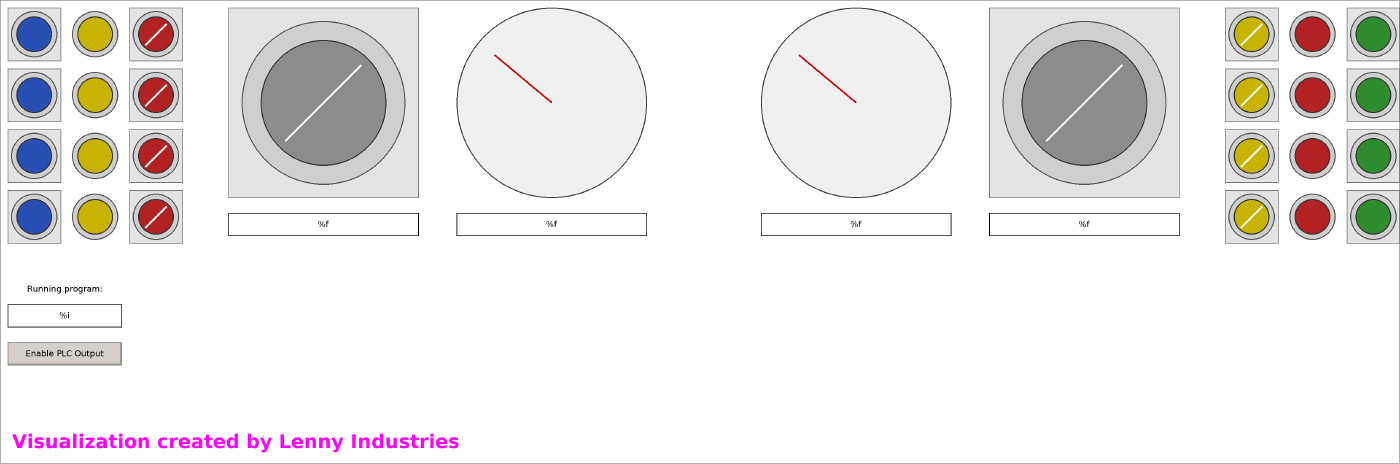
VISUALIZATION Visualization  // 1840x610
    PushSwitch (10,10 70x70), tooltip "Button 1", variable: GVL.bButton_1, behaviour: TAP, style: Switch-PushSwitch-Blue
    PushSwitch (10,90 70x70), tooltip "Button 2", variable: GVL.bButton_2, behaviour: TAP, style: Switch-PushSwitch-Blue
    PushSwitch (10,170 70x70), tooltip "Button 3", variable: GVL.bButton_3, behaviour: TAP, style: Switch-PushSwitch-Blue
    PushSwitch (10,250 70x70), tooltip "Button 4", variable: GVL.bButton_4, behaviour: TAP, style: Switch-PushSwitch-Blue
    Lamp1 (90,10 70x70), tooltip "Lamp 1", variable: GVL.bLamp_1, style: Lamp-Lamp1-Yellow
    Lamp1 (90,90 70x70), tooltip "Lamp 2", variable: GVL.bLamp_2, style: Lamp-Lamp1-Yellow
    Lamp1 (90,170 70x70), tooltip "Lamp 3", variable: GVL.bLamp_3, style: Lamp-Lamp1-Yellow
    Lamp1 (90,250 70x70), tooltip "Lamp 4", variable: GVL.bLamp_4, style: Lamp-Lamp1-Yellow
    RotarySwitch (170,10 70x70), tooltip "Switch 1", variable: GVL.bSwitch_1, behaviour: TOGGLE, style: Switch-RotarySwitch-Red
    RotarySwitch (170,90 70x70), tooltip "Switch 2", variable: GVL.bSwitch_2, behaviour: TOGGLE, style: Switch-RotarySwitch-Red
    RotarySwitch (170,170 70x70), tooltip "Switch 3", variable: GVL.bSwitch_3, behaviour: TOGGLE, style: Switch-RotarySwitch-Red
    RotarySwitch (170,250 70x70), tooltip "Switch 4", variable: GVL.bSwitch_4, behaviour: TOGGLE, style: Switch-RotarySwitch-Red
    Meter360 (600,10 250x250), value: GVL.fMeter_1, style: Meter-Meter360-Gray, scale format: %.1f, scale -200..1000
    Potentiometer360 (300,10 250x250), variable: GVL.fPotentiometer_1, style: Potentiometer-Potentiometer360-Gray, scale format: %.1f, scale 0..10
    Rectangle (300,280 250x30), "%f", tooltip "Click to change", text variable: GVL.fPotentiometer_1
        OnMouseDown: write the text variable via VisuDialogs.Numpad, min 0, max 10, format %f
    Rectangle (600,280 250x30), "%f", text variable: GVL.fMeter_1
    Label (10,550 600x60), "Visualization created by Lenny Industries"
    Meter360 (1000,10 250x250), value: GVL.fMeter_2, style: Meter-Meter360-Gray, scale format: %.1f, scale 0..100
    Potentiometer360 (1300,10 250x250), variable: GVL.fPotentiometer_2, style: Potentiometer-Potentiometer360-Gray, scale format: %.1f, scale 0..10
    Rectangle (1300,280 250x30), "%f", tooltip "Click to change", text variable: GVL.fPotentiometer_2
        OnMouseDown: write the text variable via VisuDialogs.Numpad, min 0, max 10, format %f
    Rectangle (1000,280 250x30), "%f", text variable: GVL.fMeter_2
    PushSwitch (1770,10 70x70), tooltip "Button 5", variable: GVL.bButton_5, behaviour: TAP, style: Switch-PushSwitch-Green
    PushSwitch (1770,90 70x70), tooltip "Button 6", variable: GVL.bButton_6, behaviour: TAP, style: Switch-PushSwitch-Green
    PushSwitch (1770,170 70x70), tooltip "Button 7", variable: GVL.bButton_7, behaviour: TAP, style: Switch-PushSwitch-Green
    PushSwitch (1770,250 70x70), tooltip "Button 8", variable: GVL.bButton_8, behaviour: TAP, style: Switch-PushSwitch-Green
    Lamp1 (1690,10 70x70), tooltip "Lamp 5", variable: GVL.bLamp_5, style: Lamp-Lamp1-Red
    Lamp1 (1690,90 70x70), tooltip "Lamp 6", variable: GVL.bLamp_6, style: Lamp-Lamp1-Red
    Lamp1 (1690,170 70x70), tooltip "Lamp 7", variable: GVL.bLamp_7, style: Lamp-Lamp1-Red
    Lamp1 (1690,250 70x70), tooltip "Lamp 8", variable: GVL.bLamp_8, style: Lamp-Lamp1-Red
    RotarySwitch (1610,10 70x70), tooltip "Switch 5", variable: GVL.bSwitch_5, behaviour: TOGGLE, style: Switch-RotarySwitch-Yellow
    RotarySwitch (1610,90 70x70), tooltip "Switch 6", variable: GVL.bSwitch_6, behaviour: TOGGLE, style: Switch-RotarySwitch-Yellow
    RotarySwitch (1610,170 70x70), tooltip "Switch 7", variable: GVL.bSwitch_7, behaviour: TOGGLE, style: Switch-RotarySwitch-Yellow
    RotarySwitch (1610,250 70x70), tooltip "Switch 8", variable: GVL.bSwitch_8, behaviour: TOGGLE, style: Switch-RotarySwitch-Yellow
    Rectangle (10,400 150x30), "%i", tooltip "Click to change running program", text variable: GVL.nProgramID
        OnMouseDown: write the text variable via VisuDialogs.Numpad, min 0, max 65536, format %i
    Label (10,365 150x30), "Running program:"
    Button (10,450 150x30), "Enable PLC Output", tooltip "Toggles between PLC I/O or VISU I/O", colour toggle: GVL.bUsePLC
        toggle GVL.bUsePLC
END_VISUALIZATION

(* stored: Version 1.1.0.1, ProductVersion 3.1.4024.12
   Visu Visualization: Id {ad1ad401-1671-43ba-bd72-0ea2d841b40c} *)
